FUNCTION F_FileTimeToDCTimestruct : DCTIMESTRUCT
VAR_INPUT
	tTimestamp: ULINT;
END_VAR
VAR
	tULarge: T_ULARGE_INTEGER;
	tFileTime: T_FILETIME;
	newDCTime: T_DCTIME64;
	
	fbToLocal: FB_FileTimeToTzSpecificLocalTime;
	//Malay Peninsula Daylight Time
	//(UTC+08:00) Kuala Lumpur, Singapore
	tzInfo: ST_TimeZoneInformation := (bias := -480);
END_VAR

tULarge:= ULINT_TO_ULARGE(tTimestamp);
tFileTime.dwLowDateTime:= tULarge.dwLowPart;
tFileTime.dwHighDateTime:= tULarge.dwHighPart;

fbToLocal(in:= tFileTime, tzInfo:= tzInfo);
newDCTime:= FILETIME_TO_DCTIME64(fbToLocal.out);

F_FileTimeToDCTimestruct:= DCTIME64_TO_DCTIMESTRUCT(newDCTime);

END_FUNCTION

(* stored: POU F_FileTimeToDCTimestruct: Id f622a996-6031-41cc-9d5a-50390f0eadb2, SpecialFunc None *)
